SUBAPPLICATION SubApp_PC_A (* Geraet A (Station 11, 192.168.1.11): liest Input_I1 und schreibt aktiv per OPC-UA (CLIENT_1_0) auf den von Geraet B ueberwachten Knoten - 'SUB style': das Protokoll steckt im MyLib::sys-Composite (logiBUS_IXA_TO_CLIENT_OPC), nicht in der Resource des Geraets *)
  (* Standard: 61499-2; Description: Copyright (c) 2026 Meisterschulen am Ostbahnhof This program and the accompanying materials are made available under the terms of the Eclipse Public License 2.0 which is available at https://www.eclipse.org/legal/epl-2.0/ SPDX-License-Identifier: EPL-2.0 *)
  (* Version 1.0, 2026-09-02, Franz Höpfinger, Meisterschulen am Ostbahnhof, initial API and implementation and/or initial documentation *)
  PACKAGE Training_OPC_UA_SUB;
  IMPORT VV::const::OPC_UA::myOpcUaAddresses::Q1_REMOTE_WRITE;
  IMPORT logiBUS::io::DI::logiBUS_DI::Input_I1;
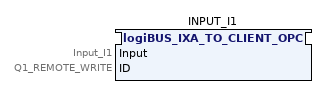
  SUBAPPS
    INPUT_I1 : MyLib::sys::logiBUS_IXA_TO_CLIENT_OPC(Input := Input_I1, ID := Q1_REMOTE_WRITE);
  END_SUBAPPS
END_SUBAPPLICATION
